% RSLogix 500 project ROLLDOOR.RSS, saved by version 8.30.00.16 %
PROJECT "ROLLDOOR"    % processor: Bul.1763 MicroLogix 1100 Series B %

PROGRAM FILES
  LAD 2   3 rungs

DATA FILES
  O0 OUTPUT  4 elements
  I1 INPUT  6 elements
  S2 STATUS  66 elements
  B3 BINARY  1 elements
  T4 TIMER  1 elements
  C5 COUNTER  1 elements
  R6 CONTROL  1 elements
  N7 INTEGER  1 elements
  F8 FLOAT  1 elements

LADDER 2
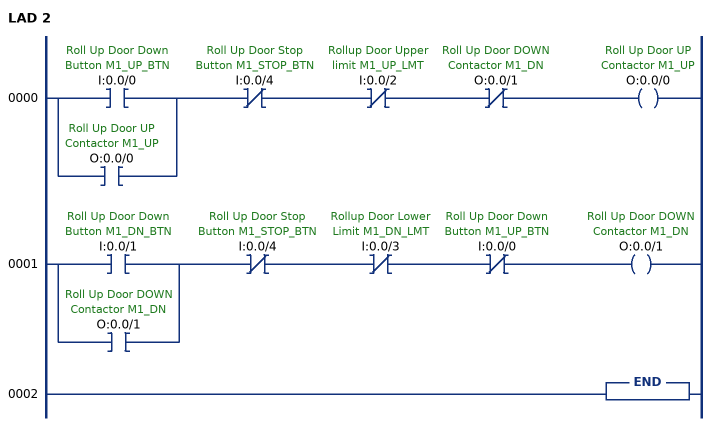
% Rung: 0 %
SOR BST XIC I:0.0/0 NXB XIC O:0.0/0 BND XIO I:0.0/4 XIO I:0.0/2 XIO O:0.0/1 OTE O:0.0/0 EOR
%   I:0.0/0  M1_UP_BTN  "Roll Up Door Down Button" %
%   O:0.0/0  M1_UP  "Roll Up Door UP Contactor" %
%   I:0.0/4  M1_STOP_BTN  "Roll Up Door Stop Button" %
%   I:0.0/2  M1_UP_LMT  "Rollup Door Upper limit" %
%   O:0.0/1  M1_DN  "Roll Up Door DOWN Contactor" %
% Rung: 1 %
SOR BST XIC I:0.0/1 NXB XIC O:0.0/1 BND XIO I:0.0/4 XIO I:0.0/3 XIO I:0.0/0 OTE O:0.0/1 EOR
%   I:0.0/1  M1_DN_BTN  "Roll Up Door Down Button" %
%   O:0.0/1  M1_DN  "Roll Up Door DOWN Contactor" %
%   I:0.0/4  M1_STOP_BTN  "Roll Up Door Stop Button" %
%   I:0.0/3  M1_DN_LMT  "Rollup Door Lower Limit" %
%   I:0.0/0  M1_UP_BTN  "Roll Up Door Down Button" %
% Rung: 2 %
SOR END EOR
